// TwinCAT 3 PLC project SYC
// ProgramVersion: 3.1.4023.0
// libraries:
//   Tc2_Standard, * (Beckhoff Automation GmbH)
//   Tc2_System, * (Beckhoff Automation GmbH)
//   Tc2_Utilities, * (Beckhoff Automation GmbH)
//   Tc3_JsonXml, * (Beckhoff Automation GmbH)
//   Tc3_Module, * (Beckhoff Automation GmbH)
//   Base Interfaces,newest,System
// project tree:
//   / Class Diagram.TcCD (not stored), MAIN.TcPOU, PlcTask.TcTTO, Testing.TcPOU
//   Collection/ HashMap.TcPOU, Map.TcIO, MutableArray.TcPOU, List.TcIO, ListLength.TcDUT (not stored), ListType.TcDUT
//   Condition/ CResult.TcDUT, Is.TcPOU
//   Misc/ AddLeadingZeros.TcPOU, BaseConnector.TcPOU, CHAR.TcDUT, CONSTANTS.TcGVL, WCHAR.TcDUT, P2CHAR.TcPOU, P2WCHAR.TcPOU
//   Sequencer/ Condition.TcPOU, Sequencer.TcPOU, StepAction.TcDUT, StepCondition.TcDUT, StepTransition.TcDUT, Transition.TcPOU
//   Sequencer/WIP/ ConditionConfig.TcDUT (not stored), CurrentStep.TcDUT (not stored), E_Result.TcTLEO, StepConfig.TcDUT, StepLog.TcDUT, StepStatus.TcDUT
//   Signal/ Signal.TcPOU, SignalBundle.TcPOU, SignalMapping.TcDUT, SignalProvider.TcPOU, SignalTimer.TcDUT
//   SimpleStepLogger/ SimpleStepLog.TcDUT, SimpleStepLogger.TcPOU
//   SymbolProvider/ Symbol.TcDUT, SymbolProvider.TcPOU, SymbolProvider_1.TcPOU
//   Tools/ CallThisSingleTimeEachCycle.TcPOU, TaskHeartbeat.TcPOU, Regex.TcPOU, RegexMatch.TcDUT, System.TcPOU, SystemBundle.TcPOU, WRegex.TcPOU, TimeProvider.TcPOU
// real-time tasks:
//   TASK PlcTask: cycle T#10ms, priority 20, ADS port 350

CONFIGURATION SYC
    RESOURCE PLC ON TwinCAT3
        TASK PlcTask(INTERVAL := T#10ms, PRIORITY := 20);
        PROGRAM MAIN WITH PlcTask : MAIN;
        PROGRAM Testing WITH PlcTask : Testing;
    END_RESOURCE
END_CONFIGURATION

// ---- Condition/CResult.TcDUT
TYPE CResult :
STRUCT
	datatype	: INT;
	result		: BOOL;
END_STRUCT
END_TYPE

// ---- Collection/ListType.TcDUT

TYPE ListType :
STRUCT
	size			: UDINT;
	class			: __SYSTEM.TYPE_CLASS;
//	classPointer	: POINTER TO BYTE; // pointer to FB
	name			: T_MaxString;

	
	(*
	IDEA:
	if __SYSTEM.TYPE_CLASS <> USER_DEF then //int, bool, string
		classNumber := __SYSTEM.TYPE_CLASS
	else // function block
		classNumber := ADR(type)
		
	problems:
	 - how to achieve this in some user firendly way
	 - how to keep datatype pointer up to date after online change
	*)
//	classNumber		: UXINT; 

END_STRUCT
END_TYPE

// ---- Misc/CHAR.TcDUT
TYPE CHAR : STRING(1); END_TYPE

// ---- Misc/WCHAR.TcDUT
TYPE WCHAR : WSTRING(1); END_TYPE

// ---- Sequencer/StepAction.TcDUT
TYPE StepAction :
STRUCT
	name			: STRING;
	caseNumber		: INT;
//	timeout			: TIME;
//	timeoutAction	: STRING; these will go to binding
	description		: STRING;
END_STRUCT
END_TYPE

// ---- Sequencer/StepCondition.TcDUT
TYPE StepCondition :
STRUCT
	name			: STRING;
	condition		: Condition;
//	nextAction		: STRING;
//	timeout			: TIME;
//	timeoutAction	: STRING;
	/// these will go to binding
END_STRUCT
END_TYPE

// ---- Sequencer/StepTransition.TcDUT
TYPE StepTransition :
STRUCT
	actionName		: STRING;
	conditionName	: STRING;
	nextActionName	: STRING;
END_STRUCT
END_TYPE

// ---- Sequencer/WIP/E_Result.TcTLEO
{attribute 'qualified_only'}
{attribute 'strict'}
TYPE E_Result :
(
	done,
	timeout,
	error,
	interrupt,
	stop
);
END_TYPE

// ---- Sequencer/WIP/StepConfig.TcDUT
TYPE StepConfig :
STRUCT
	number		: INT;
	timeout		: TIME;
	
	description	: STRING;
END_STRUCT
END_TYPE

// ---- Sequencer/WIP/StepLog.TcDUT
TYPE StepLog :
STRUCT
	config 		: StepConfig;
	status		: StepStatus;
END_STRUCT
END_TYPE

// ---- Sequencer/WIP/StepStatus.TcDUT
TYPE StepStatus :
STRUCT
	status		: E_Result;
	elapsedTime : TIME;
END_STRUCT
END_TYPE

// ---- Signal/SignalMapping.TcDUT
TYPE SignalMapping :
STRUCT
	symbol	: POINTER TO BOOL;
	signal	: POINTER TO SignalBundle;
END_STRUCT
END_TYPE

// ---- Signal/SignalTimer.TcDUT

// Basically just timer IO with IN input excluded as it binded to the signal variable
TYPE SignalTimer :
STRUCT
	PT		: REFERENCE TO TIME;
	
	ET		: REFERENCE TO TIME;
	Q		: REFERENCE TO BOOL;
END_STRUCT
END_TYPE

// ---- SimpleStepLogger/SimpleStepLog.TcDUT
TYPE SimpleStepLog :
STRUCT
	number			: LINT;
	name			: STRING;
	description		: T_MaxString;
	duration		: TIME;
	mode			: STRING;
END_STRUCT
END_TYPE

// ---- SymbolProvider/Symbol.TcDUT
TYPE Symbol :
STRUCT
	info : __SYSTEM.AnyType; // varinfo?
	
	description : STRING;
END_STRUCT
END_TYPE

// ---- Tools/RegexMatch.TcDUT
TYPE RegexMatch :
STRUCT
	found : BOOL;
	start : INT;
	length : INT;
	text : STRING;
END_STRUCT
END_TYPE

// ---- Misc/CONSTANTS.TcGVL
VAR_GLOBAL CONSTANT
	MAX_DWORD	: DWORD := 4294967295;
	MAX_DWORD_2	: DWORD := -1;
	MAX_TIME	: TIME := TO_TIME(MAX_DWORD);
END_VAR

// ---- Collection/Map.TcIO

INTERFACE Map


METHOD Get : BOOL
VAR_INPUT
	
END_VAR
END_METHOD


METHOD Put : Map
VAR_INPUT
	key			: ANY;
	value		: ANY;
END_VAR
END_METHOD


METHOD Remove : Map
VAR_INPUT
END_VAR
END_METHOD


METHOD RemoveAll : Map
VAR_INPUT
END_VAR
END_METHOD

END_INTERFACE

// ---- Collection/List.TcIO

INTERFACE List


METHOD Append : List
VAR_INPUT
	data	: ANY;
END_VAR
END_METHOD


PROPERTY Datatype : ListType
GET
END_GET
END_PROPERTY

PROPERTY DatatypeDefined : BOOL
GET
END_GET
END_PROPERTY


// Delete pointers
METHOD FB_exit : BOOL
VAR_INPUT
	bInCopyCode : BOOL; // if TRUE, the exit method is called for exiting an instance that is copied afterwards (online change).
END_VAR
END_METHOD


METHOD Get : BOOL
VAR_INPUT
	index		: INT; // Allow for indexing from end
	destination	: ANY;
END_VAR
END_METHOD


METHOD Insert : List
VAR_INPUT
	index	: INT; // Allow for indexing from end
	data	: ANY;
END_VAR
END_METHOD


METHOD IsEmpty : BOOL
VAR_INPUT
END_VAR
END_METHOD


METHOD IsTypeCorrect : BOOL
VAR_INPUT
	checkedVariable		: ANY;
END_VAR
END_METHOD


PROPERTY LastIndex : ListLength
GET
END_GET
END_PROPERTY


PROPERTY Length : ListLength
GET
END_GET
END_PROPERTY


METHOD Prepend : List
VAR_INPUT
	data	: ANY;
END_VAR
END_METHOD


METHOD Remove : List
VAR_INPUT
	index	: INT; // Allow for indexing from end
END_VAR
END_METHOD


METHOD RemoveAll : List
VAR_INPUT
END_VAR
END_METHOD


METHOD Set : List
VAR_INPUT
	index	: INT; // Allow for indexing from end
	data	: ANY;
END_VAR
END_METHOD

END_INTERFACE

// ---- MAIN.TcPOU
PROGRAM MAIN
VAR
	sensor1 : BOOL;
	sensor2 : BOOL;
	sensor3 : BOOL;
	counter1 : INT;
	
	seq : Sequencer;
	firstCycle : BOOL := TRUE;
	test : BOOL;
	ceres : CResult;
	n1 : PVOID;
	n2 : PVOID;
	n3 : PVOID;
	
	re : Regex;
END_VAR

IF firstCycle THEN
	firstCycle := FALSE;
	
	RegisterActions();
	
END_IF

seq();

CASE seq.currentAction.caseNumber OF
	0 : // action code 1
	10 : // action code 2
	20 : // action code 3
	30 : // action code 4

END_CASE

Is(test);
Is(ceres);

n1 := SIZEOF(CResult);
n2 := SIZEOF(CResult.result);
n3 := SIZEOF(CResult.datatype);

re.match(pattern := 'he.*o', text := 'hellQQllo_HelloWorld').found;

ACTION RegisterActions:
//seq.ClearActions();

//seq.RegisterAction(
//	name := 'name 1',
//	number := 0
//);
//seq.RegisterAction(
//	name := 'name 2',
//	number := 10
//);
//seq.RegisterAction(
//	name := 'name 3',
//	number := 20
//);
//seq.RegisterAction(
//	name := 'name 4',
//	number := 30
//);
END_ACTION

ACTION RegisterAll:
// Register actions
seq.RegisterAction(
	name := 'name 1',
	caseNumber := 0,
	''
);
seq.RegisterAction(
	name := 'name 2',
	caseNumber := 10,
	''
);
seq.RegisterAction(
	name := 'name 3',
	caseNumber := 20,
	''
);
seq.RegisterAction(
	name := 'name 4',
	caseNumber := 30,
	''
);

// Register conditions
seq.RegisterCondition('cond 1').Is(sensor1);
seq.RegisterCondition('cond 2').Is(sensor2).AndIs(sensor3);
seq.RegisterCondition('cond 3').Is(sensor3);
seq.RegisterCondition('cond 4').Is(sensor3);

// Bind them together
seq.Bind('name 1')
	.WhenGoTo('cond 1', 'name 2');
seq.Bind('name 2')
	.WhenGoTo('cond 2', 'name 3')
	.WhenGoTo('cond 3', 'name 4');
seq.Bind('name 3')
	.WhenGoTo('cond 3', 'name 4');
seq.Bind('name 4')
	.WhenGoTo('cond 4', 'name 1');
END_ACTION

ACTION RegisterConditions:
//seq.ClearConditions();

//seq.RegisterCondition('cond 1').Is(sensor1);
//seq.RegisterCondition('cond 2').Is(sensor2).AndIs(sensor3);
//seq.RegisterCondition('cond 3').Is(sensor3);
//seq.RegisterCondition('cond 4').Is(sensor3);
END_ACTION

ACTION RegisterTransitions:
//seq.Bind('name 1')
//	.WhenGoTo('cond 1', 'name 2');
//seq.Bind('name 2')
//	.WhenGoTo('cond 2', 'name 3')
//	.WhenGoTo('cond 3', 'name 4');
//seq.Bind('name 3')
//	.WhenGoTo('cond 3', 'name 4');
//seq.Bind('name 4')
//	.WhenGoTo('cond 4', 'name 1');
END_ACTION

END_PROGRAM

// ---- Sequencer/Sequencer.TcPOU
FUNCTION_BLOCK Sequencer EXTENDS BaseConnector
VAR_INPUT
END_VAR
VAR_OUTPUT
END_VAR
VAR
	actions		: ARRAY[0..MAX_ACTION] OF StepAction;
	lastAction 	: INT := 0;
	currentAction : StepAction;
	startAction	: STRING;
	
	conditions	: ARRAY[0..MAX_CONDITION] OF StepCondition;
	lastCondition : INT := 0;
	currentCondition : StepCondition;
	
	timer		: TON := (PT := MAX_TIME);
	
END_VAR
VAR CONSTANT
	MAX_ACTION	: INT := 99;
	MAX_CONDITION : INT := 99;
END_VAR


timer(IN := TRUE);

//IF currentCondition.condition.satisfied THEN
	
//	ChangeStep(currentCondition.nextAction);
//ELSIF currentAction.timeout > T#0S AND_THEN timer.ET > currentAction.timeout THEN
	
//	ChangeStep(currentAction.timeoutAction);
//ELSIF currentCondition.timeout > T#0S AND_THEN timer.ET > currentCondition.timeout THEN

//	ChangeStep(currentCondition.timeoutAction);
//END_IF

METHOD Bind : REFERENCE TO Transition
VAR_INPUT
	actionName	: STRING;
END_VAR
END_METHOD

METHOD ChangeStep : BOOL
VAR_INPUT
	actionName		: STRING;
END_VAR
VAR
	i : INT;
END_VAR
//LogChange(currentAction.name, Condition, actionName);

FOR i := 0 TO MAX_ACTION DO
	IF (actions[i].name = actionName) THEN
		
		currentAction := actions[i];
	END_IF
END_FOR

timer(IN := FALSE);
timer(IN := TRUE);
END_METHOD

METHOD PRIVATE LogChange : BOOL
VAR_INPUT
	oldAction : STRING;
	satisfiedCondition : Condition;
	nextAction : STRING;
END_VAR
// TODO
END_METHOD

METHOD RegisterAction : BOOL
VAR_INPUT
	name			: STRING;
	caseNumber		: INT;
	description		: STRING;
END_VAR
VAR
	a : REFERENCE TO StepAction REF= actions[lastAction];
END_VAR
a.name := name;
a.caseNumber := caseNumber;
//a.timeout := timeout;
//a.timeoutAction := timeoutAction;
a.description := description;

lastAction := lastAction + 1;
END_METHOD

METHOD RegisterCondition : REFERENCE TO Condition
VAR_INPUT
	name			: STRING;
END_VAR
VAR
	c : REFERENCE TO StepCondition REF= conditions[lastAction];
END_VAR
c.name := name;
//c.condition := condition;
//c.nextAction := nextAction;
//c.timeout := timeout;
//c.timeoutAction := timeoutAction;

lastCondition := lastCondition + 1;

RegisterCondition REF= c.condition;
END_METHOD

METHOD Start : BOOL
VAR_INPUT
	startAction		: STRING;
END_VAR
THIS^.startAction := startAction; 

ChangeStep(startAction);
END_METHOD

END_FUNCTION_BLOCK

// ---- Misc/BaseConnector.TcPOU
FUNCTION_BLOCK BaseConnector
VAR_INPUT
END_VAR
VAR_OUTPUT
END_VAR
VAR
END_VAR
VAR_STAT
	sp	: SymbolProvider;
END_VAR

END_FUNCTION_BLOCK

// ---- SymbolProvider/SymbolProvider.TcPOU
FUNCTION_BLOCK SymbolProvider
VAR_INPUT
END_VAR
VAR_OUTPUT
END_VAR
VAR
	list : ARRAY[0..99] OF Symbol;
	lastIndex : UINT := 0;
END_VAR

METHOD Get : STRING
VAR_INPUT
	symbol : ANY;
END_VAR
VAR
	i : UINT;
END_VAR
FOR i := 0 TO lastIndex DO
	IF symbol.pValue = list[i].info.pValue THEN
		Get := list[i].description;
		RETURN;
	END_IF
END_FOR
END_METHOD

METHOD Register : BOOL
VAR_INPUT
	symbol				: ANY;
	descriptionName		: STRING;
END_VAR
list[lastIndex].info := symbol;
list[lastIndex].description := descriptionName;
END_METHOD

END_FUNCTION_BLOCK

// ---- Sequencer/Transition.TcPOU
FUNCTION_BLOCK Transition
VAR_INPUT
END_VAR
VAR_OUTPUT
END_VAR
VAR
END_VAR

METHOD WhenGoTo : reference TO Transition
VAR_INPUT
	conditionName	: STRING;
	nextActionName	: STRING;
END_VAR
END_METHOD

END_FUNCTION_BLOCK

// ---- Sequencer/Condition.TcPOU
FUNCTION_BLOCK Condition EXTENDS BaseConnector
VAR_INPUT
END_VAR
VAR_OUTPUT
END_VAR
VAR
	config		: ARRAY[0..99] OF ConditionConfig;
	result		: BOOL;
END_VAR

METHOD AndIs : REFERENCE TO Condition
VAR_INPUT
	symbol	: ANY;
END_VAR
END_METHOD

METHOD AndIsNot : Condition
VAR_INPUT
END_VAR
END_METHOD

METHOD Is : REFERENCE TO Condition
VAR_INPUT
	symbol	: ANY;
END_VAR
END_METHOD

METHOD IsNot : Condition
VAR_INPUT
END_VAR
END_METHOD

METHOD OrIs : Condition
VAR_INPUT
END_VAR
END_METHOD

METHOD OrIsNot : Condition
VAR_INPUT
END_VAR
END_METHOD

PROPERTY satisfied : BOOL
GET
END_GET
END_PROPERTY

END_FUNCTION_BLOCK

// ---- Condition/Is.TcPOU
FUNCTION Is : CResult
VAR_INPUT
	symbol		: ANY;
END_VAR
VAR
	typeReader	: FB_JsonReadWriteDatatype;
	t : STRING;
END_VAR

CASE symbol.TypeClass OF
	
	IBaseLibrary.TypeClass.TYPE_BOOL:

		Is.result := PBOOL_TO_BOOL(symbol.pValue);
		Is.datatype := TO_INT(symbol.TypeClass);
		
	IBaseLibrary.TypeClass.TYPE_USERDEF:
		IF typeReader.GetDatatypeNameByAddress(pData := symbol.pValue, nData := symbol.diSize) = 'CResult' THEN

			Is.result := PBOOL_TO_BOOL(symbol.pValue + ADR(Is.result) - ADR(Is));
			Is.datatype := 420;
		END_IF

END_CASE

END_FUNCTION

// ---- Tools/Regex.TcPOU
FUNCTION_BLOCK Regex
VAR_INPUT
END_VAR
VAR_OUTPUT
END_VAR
VAR
	result : RegexMatch;
END_VAR

//https://stackoverflow.com/questions/4040835/how-do-i-write-a-simple-regular-expression-pattern-matching-function-in-c-or-c

METHOD incMatchPos : BOOL
VAR_INPUT
	isMatch : BOOL;
END_VAR
IF isMatch THEN
	result.length := result.length + 1;
ELSE
	result.start := result.start + 1;
	result.length := 0;
END_IF
incMatchPos := isMatch;
END_METHOD

METHOD match : REFERENCE TO RegexMatch
VAR_INPUT
	pattern : STRING;
	text	: STRING;
END_VAR
result.start := 1;
result.length := 0;
result.found := matchP(ADR(pattern), ADR(text));
result.text := MID(STR := text, POS := result.start, LEN := result.length);

match REF= result;
END_METHOD

METHOD PRIVATE matchHere : BOOL
VAR_INPUT
	pattern : POINTER TO STRING;
	text	: POINTER TO STRING;
END_VAR
IF P2CHAR(pattern) = '$00' THEN
	matchHere := TRUE;
	RETURN;
ELSIF P2CHAR(pattern + 1) = '*' THEN
	matchHere := matchStar(P2CHAR(pattern), pattern + 2, text);
	RETURN;
ELSIF P2CHAR(pattern) = '$$' AND P2CHAR(pattern + 1) = '$00' THEN
	matchHere := P2CHAR(text) = '$00';
	RETURN;
ELSIF text^ <> '$00' AND (P2CHAR(pattern) = '.' OR P2CHAR(pattern) = P2CHAR(text)) THEN
	matchHere := THIS^.matchHere(pattern + 1, text + 1);
	incMatchPos(matchHere);
	RETURN;
END_IF



///* matchhere: search FOR regexp AT beginning OF text */
//int matchhere(char *regexp, char *text)
//{
//    if (regexp[0] == '\0')
//        return 1;
//    if (regexp[1] == '*')
//        return matchstar(regexp[0], regexp+2, text);
//    if (regexp[0] == '$' && regexp[1] == '\0')
//        return *text == '\0';
//    if (*text!='\0' && (regexp[0]=='.' || regexp[0]==*text))
//        return matchhere(regexp+1, text+1);
//    return 0;
//}
END_METHOD

METHOD matchP : BOOL
VAR_INPUT
	pattern : POINTER TO STRING;
	text	: POINTER TO STRING;
END_VAR
IF P2CHAR(pattern) = '^' THEN
	matchP := matchHere(pattern + 1, text);
	RETURN;
END_IF
REPEAT
	IF matchHere(pattern, text) THEN
		matchP := TRUE;
		RETURN;
	END_IF
UNTIL
	NOT(P2CHAR(text) <> '$00') AND (text := text + 1) <> NULL AND (incMatchPos(matchP) OR TRUE) //pointer dereference and increment oneliner
END_REPEAT



///* match: search FOR regexp anywhere in text */
//int match(char *regexp, char *text)
//{
//    if (regexp[0] == '^')
//        return matchhere(regexp+1, text);
//    do {    /* must look even if string is empty */
//        if (matchhere(regexp, text))
//            return 1;
//    } while (*text++ != '\0');
//    return 0;
//}
END_METHOD

METHOD PRIVATE matchStar : BOOL
VAR_INPUT
	c		: CHAR;
	pattern : POINTER TO STRING;
	text	: POINTER TO STRING;
END_VAR
REPEAT
	IF matchHere(pattern, text) THEN
		matchStar := TRUE;
		RETURN;
	END_IF
UNTIL
	NOT(P2CHAR(text) <> '$00' AND (P2CHAR(text) = c OR c = '.')) AND (text := text + 1) > null AND (incMatchPos(NOT matchStar) OR TRUE)
END_REPEAT


///* matchstar: search FOR c*regexp AT beginning OF text */
//int matchstar(int c, char *regexp, char *text)
//{
//    do {    /* a * matches zero or more instances */
//        if (matchhere(regexp, text))
//            return 1;
//    } while (*text != '\0' && (*text++ == c || c == '.'));
//    return 0;
//}
END_METHOD

END_FUNCTION_BLOCK

// ---- Misc/P2CHAR.TcPOU
FUNCTION P2CHAR : CHAR
VAR_INPUT
	p : POINTER TO STRING;
END_VAR
VAR
END_VAR

P2CHAR := p^;

END_FUNCTION

// ---- Testing.TcPOU
PROGRAM Testing
VAR
	test		: STRING := 'ahoj';
	byteContent	: ARRAY[1..SIZEOF(test)] OF BYTE;
	
	beat : BOOL;
	t : STRING;
END_VAR

test := TO_STRING(ADR(byteContent));

CallThisSingleTimeEachCycle();


beat := System().GetTaskHeartbeat();
t := System().TimeProvider.GetTimeString('{h}:{m}:{s},{S}');

END_PROGRAM

// ---- Tools/CallThisSingleTimeEachCycle.TcPOU

FUNCTION CallThisSingleTimeEachCycle : BOOL


TaskHeartbeat(update := TRUE);

END_FUNCTION

// ---- Tools/TaskHeartbeat.TcPOU

FUNCTION TaskHeartbeat : BOOL;
VAR_INPUT
	update		: BOOL;
END_VAR
VAR_STAT
	_beat		: BOOL;
END_VAR


IF (update) THEN
	_beat := NOT _beat;
END_IF

TaskHeartbeat := _beat;

END_FUNCTION

// ---- Tools/System.TcPOU

FUNCTION System : REFERENCE TO SystemBundle
VAR_INPUT
END_VAR
VAR
	bundle		: SystemBundle;
END_VAR


bundle.Call();

System REF= bundle;

END_FUNCTION

// ---- Tools/SystemBundle.TcPOU

FUNCTION_BLOCK SystemBundle
VAR_INPUT
END_VAR
VAR_OUTPUT
END_VAR
VAR
	_timeProvider		: TimeProvider;
END_VAR

METHOD Call : BOOL
VAR_INPUT
END_VAR

_timeProvider();
END_METHOD


METHOD GetTaskHeartbeat : BOOL
VAR_INPUT
END_VAR

GetTaskHeartbeat := TaskHeartbeat(update := FALSE);
END_METHOD

PROPERTY TimeProvider : REFERENCE TO TimeProvider
GET

TimeProvider REF= _timeProvider;
END_GET
END_PROPERTY

END_FUNCTION_BLOCK

// ---- Tools/TimeProvider.TcPOU
FUNCTION_BLOCK TimeProvider
VAR_INPUT
END_VAR
VAR_OUTPUT
END_VAR
VAR
	localSystemTime						: FB_LocalSystemTime;
	
	// timestamp
	getTimeZoneInformation 			: FB_GetTimeZoneInformation;
    timeZoneInformation 			: ST_TimeZoneInformation;
    specificLocalTimeToFileTime 	: FB_TzSpecificLocalTimeToFileTime;
    fileTime						: T_FILETIME;
    onZerothSecondLastCycle 		: BOOL;
END_VAR

localSystemTime(bEnable := FALSE);


//https://stackoverflow.com/questions/41773732/how-do-i-get-the-unix-timestamp-in-twincat3

// On the zeroth second of each minutesync timezone information
IF (timeZoneInformation.standardName = '' OR (localSystemTime.systemTime.wSecond = 0 AND NOT onZerothSecondLastCycle)) THEN
    getTimeZoneInformation(sNetID := '', bExecute := TRUE, tzInfo => timeZoneInformation);
END_IF;

// Convert local system time to unix timestamps
specificLocalTimeToFileTime(in := Tc2_Utilities.SYSTEMTIME_TO_FILETIME(localSystemTime.systemTime), tzInfo := timeZoneInformation, out => fileTime);
//seconds := (SHL(DWORD_TO_ULINT(fileTime.dwHighDateTime), 32) + DWORD_TO_ULINT(fileTime.dwLowDateTime)) / 10000000 - 11644473600;
//milliseconds := (SHL(DWORD_TO_ULINT(fileTime.dwHighDateTime), 32) + DWORD_TO_ULINT(fileTime.dwLowDateTime)) / 10000 - 11644473600000;

onZerothSecondLastCycle := localSystemTime.systemTime.wSecond = 0;

METHOD FB_init : BOOL
VAR_INPUT
	bInitRetains : BOOL; // if TRUE, the retain variables are initialized (warm start / cold start)
	bInCopyCode : BOOL;  // if TRUE, the instance afterwards gets moved into the copy code (online change)
END_VAR
localSystemTime(bEnable := TRUE);
END_METHOD

METHOD GetMonthName : STRING
VAR_INPUT
	monthNumber			: UINT;
	shortName			: BOOL;
END_VAR
IF shortName THEN
	CASE monthNumber OF
		1	: GetMonthName := 'Jan';
		2	: GetMonthName := 'Feb';
		3	: GetMonthName := 'Mar';
		4	: GetMonthName := 'Apr';
		5	: GetMonthName := 'May';
		6	: GetMonthName := 'Jun';
		7	: GetMonthName := 'Jul';
		8	: GetMonthName := 'Aug';
		9	: GetMonthName := 'Sep';
		10	: GetMonthName := 'Oct';
		11	: GetMonthName := 'Nov';
		12	: GetMonthName := 'Dec';
	END_CASE
ELSE
	CASE monthNumber OF
		1	: GetMonthName := 'January';
		2	: GetMonthName := 'February';
		3	: GetMonthName := 'March';
		4	: GetMonthName := 'April';
		5	: GetMonthName := 'May';
		6	: GetMonthName := 'June';
		7	: GetMonthName := 'July';
		8	: GetMonthName := 'August';
		9	: GetMonthName := 'September';
		10	: GetMonthName := 'October';
		11	: GetMonthName := 'November';
		12	: GetMonthName := 'December';
	END_CASE
END_IF
END_METHOD

METHOD GetTimeString : STRING
VAR_INPUT
	format : STRING; //hh:mm:ss:SSS dd:MM:yyyy https://www.ibm.com/docs/en/rtw/9.0.1?topic=reference-formatting-parsing-date-time-patterns
END_VAR
VAR
	placeholder : STRING(4);
	
	beginIndex	: INT;
	endIndex	: INT;
	length		: INT;
		
END_VAR
GetTimeString := format;

WHILE (beginIndex := FIND(GetTimeString, '{')) > 0 AND (endIndex := FIND(GetTimeString, '}')) > (beginIndex + 1) AND  (length := endIndex - beginIndex - 1) > 0 DO
	
	placeholder := MID(STR := GetTimeString, POS := beginIndex + 1, LEN := length);
		
	IF 		placeholder = 'h' 		THEN GetTimeString := REPLACE( STR1 := GetTimeString, STR2 := TO_STRING(localSystemTime.systemTime.wHour), L := length + 2, P := beginIndex);
	ELSIF 	placeholder = 'hh' 		THEN GetTimeString := REPLACE( STR1 := GetTimeString, STR2 := AddLeadingZeros(TO_STRING(localSystemTime.systemTime.wHour), 2), L := length + 2, P := beginIndex);
	ELSIF 	placeholder = 'm' 		THEN GetTimeString := REPLACE( STR1 := GetTimeString, STR2 := TO_STRING(localSystemTime.systemTime.wMinute), L := length + 2, P := beginIndex);
	ELSIF 	placeholder = 'mm' 		THEN GetTimeString := REPLACE( STR1 := GetTimeString, STR2 := AddLeadingZeros(TO_STRING(localSystemTime.systemTime.wMinute), 2), L := length + 2, P := beginIndex);
	ELSIF 	placeholder = 's' 		THEN GetTimeString := REPLACE( STR1 := GetTimeString, STR2 := TO_STRING(localSystemTime.systemTime.wSecond), L := length + 2, P := beginIndex);
	ELSIF 	placeholder = 'ss' 		THEN GetTimeString := REPLACE( STR1 := GetTimeString, STR2 := AddLeadingZeros(TO_STRING(localSystemTime.systemTime.wSecond), 2), L := length + 2, P := beginIndex);
	ELSIF 	placeholder = 'S' 		THEN GetTimeString := REPLACE( STR1 := GetTimeString, STR2 := TO_STRING(localSystemTime.systemTime.wMilliseconds/100), L := length + 2, P := beginIndex);
	ELSIF 	placeholder = 'SS' 		THEN GetTimeString := REPLACE( STR1 := GetTimeString, STR2 := AddLeadingZeros(TO_STRING(localSystemTime.systemTime.wMilliseconds/10), 2), L := length + 2, P := beginIndex);
	ELSIF 	placeholder = 'SSS' 	THEN GetTimeString := REPLACE( STR1 := GetTimeString, STR2 := AddLeadingZeros(TO_STRING(localSystemTime.systemTime.wMilliseconds), 3), L := length + 2, P := beginIndex);
	ELSIF 	placeholder = 'd' 		THEN GetTimeString := REPLACE( STR1 := GetTimeString, STR2 := TO_STRING(localSystemTime.systemTime.wDay), L := length + 2, P := beginIndex);
	ELSIF 	placeholder = 'dd' 		THEN GetTimeString := REPLACE( STR1 := GetTimeString, STR2 := AddLeadingZeros(TO_STRING(localSystemTime.systemTime.wDay), 2), L := length + 2, P := beginIndex);
	ELSIF 	placeholder = 'ddd' 	THEN GetTimeString := REPLACE( STR1 := GetTimeString, STR2 := GetWeekdayName(localSystemTime.systemTime.wDayOfWeek, TRUE), L := length + 2, P := beginIndex);
	ELSIF 	placeholder = 'dddd'	THEN GetTimeString := REPLACE( STR1 := GetTimeString, STR2 := GetWeekdayName(localSystemTime.systemTime.wDayOfWeek, FALSE), L := length + 2, P := beginIndex);
	ELSIF 	placeholder = 'M' 		THEN GetTimeString := REPLACE( STR1 := GetTimeString, STR2 := TO_STRING(localSystemTime.systemTime.wMonth), L := length + 2, P := beginIndex);
	ELSIF 	placeholder = 'MM' 		THEN GetTimeString := REPLACE( STR1 := GetTimeString, STR2 := AddLeadingZeros(TO_STRING(localSystemTime.systemTime.wMonth), 2), L := length + 2, P := beginIndex);
	ELSIF 	placeholder = 'MMM' 	THEN GetTimeString := REPLACE( STR1 := GetTimeString, STR2 := GetMonthName(localSystemTime.systemTime.wMonth, TRUE), L := length + 2, P := beginIndex);
	ELSIF 	placeholder = 'MMMM'	THEN GetTimeString := REPLACE( STR1 := GetTimeString, STR2 := GetMonthName(localSystemTime.systemTime.wMonth, FALSE), L := length + 2, P := beginIndex);
	ELSIF 	placeholder = 'y' OR placeholder = 'yy' OR placeholder = 'yyy' OR placeholder = 'yyyy'
									THEN GetTimeString := REPLACE( STR1 := GetTimeString, STR2 := RIGHT(TO_STRING(localSystemTime.systemTime.wYear), length), L := length + 2, P := beginIndex);
	ELSE 
			GetTimeString := REPLACE( STR1 := GetTimeString, STR2 := 'ERR', L := length + 2, P := beginIndex);
	END_IF
END_WHILE
END_METHOD

// deprecated. Use optimized GetTimeString() instead
METHOD GetTimeStringRe : STRING
VAR_INPUT
	format : STRING; //hh:mm:ss:SSS dd:MM:yyyy https://www.ibm.com/docs/en/rtw/9.0.1?topic=reference-formatting-parsing-date-time-patterns
END_VAR
VAR
	re : Regex;
	placeholder : STRING(4);
END_VAR
GetTimeStringRe := format;

WHILE re.match('{.*}', GetTimeStringRe).found DO
	placeholder := MID(STR := re.result.text, POS := 2, LEN := re.result.length - 2);
	
	IF 		placeholder = 'h' 		THEN GetTimeStringRe := REPLACE( STR1 := GetTimeStringRe, STR2 := TO_STRING(localSystemTime.systemTime.wHour), L := re.result.length, P := re.result.start);
	ELSIF 	placeholder = 'hh' 		THEN GetTimeStringRe := REPLACE( STR1 := GetTimeStringRe, STR2 := AddLeadingZeros(TO_STRING(localSystemTime.systemTime.wHour), 2), L := re.result.length, P := re.result.start);
	ELSIF 	placeholder = 'm' 		THEN GetTimeStringRe := REPLACE( STR1 := GetTimeStringRe, STR2 := TO_STRING(localSystemTime.systemTime.wMinute), L := re.result.length, P := re.result.start);
	ELSIF 	placeholder = 'mm' 		THEN GetTimeStringRe := REPLACE( STR1 := GetTimeStringRe, STR2 := AddLeadingZeros(TO_STRING(localSystemTime.systemTime.wMinute), 2), L := re.result.length, P := re.result.start);
	ELSIF 	placeholder = 's' 		THEN GetTimeStringRe := REPLACE( STR1 := GetTimeStringRe, STR2 := TO_STRING(localSystemTime.systemTime.wSecond), L := re.result.length, P := re.result.start);
	ELSIF 	placeholder = 'ss' 		THEN GetTimeStringRe := REPLACE( STR1 := GetTimeStringRe, STR2 := AddLeadingZeros(TO_STRING(localSystemTime.systemTime.wSecond), 2), L := re.result.length, P := re.result.start);
	ELSIF 	placeholder = 'S' 		THEN GetTimeStringRe := REPLACE( STR1 := GetTimeStringRe, STR2 := TO_STRING(localSystemTime.systemTime.wMilliseconds/100), L := re.result.length, P := re.result.start);
	ELSIF 	placeholder = 'SS' 		THEN GetTimeStringRe := REPLACE( STR1 := GetTimeStringRe, STR2 := AddLeadingZeros(TO_STRING(localSystemTime.systemTime.wMilliseconds/10), 2), L := re.result.length, P := re.result.start);
	ELSIF 	placeholder = 'SSS' 	THEN GetTimeStringRe := REPLACE( STR1 := GetTimeStringRe, STR2 := AddLeadingZeros(TO_STRING(localSystemTime.systemTime.wMilliseconds), 3), L := re.result.length, P := re.result.start);
	ELSIF 	placeholder = 'd' 		THEN GetTimeStringRe := REPLACE( STR1 := GetTimeStringRe, STR2 := TO_STRING(localSystemTime.systemTime.wDay), L := re.result.length, P := re.result.start);
	ELSIF 	placeholder = 'dd' 		THEN GetTimeStringRe := REPLACE( STR1 := GetTimeStringRe, STR2 := AddLeadingZeros(TO_STRING(localSystemTime.systemTime.wDay), 2), L := re.result.length, P := re.result.start);
	ELSIF 	placeholder = 'ddd' 	THEN GetTimeStringRe := REPLACE( STR1 := GetTimeStringRe, STR2 := GetWeekdayName(localSystemTime.systemTime.wDayOfWeek, TRUE), L := re.result.length, P := re.result.start);
	ELSIF 	placeholder = 'dddd'	THEN GetTimeStringRe := REPLACE( STR1 := GetTimeStringRe, STR2 := GetWeekdayName(localSystemTime.systemTime.wDayOfWeek, FALSE), L := re.result.length, P := re.result.start);
	ELSIF 	placeholder = 'M' 		THEN GetTimeStringRe := REPLACE( STR1 := GetTimeStringRe, STR2 := TO_STRING(localSystemTime.systemTime.wMonth), L := re.result.length, P := re.result.start);
	ELSIF 	placeholder = 'MM' 		THEN GetTimeStringRe := REPLACE( STR1 := GetTimeStringRe, STR2 := AddLeadingZeros(TO_STRING(localSystemTime.systemTime.wMonth), 2), L := re.result.length, P := re.result.start);
	ELSIF 	placeholder = 'MMM' 	THEN GetTimeStringRe := REPLACE( STR1 := GetTimeStringRe, STR2 := GetMonthName(localSystemTime.systemTime.wMonth, TRUE), L := re.result.length, P := re.result.start);
	ELSIF 	placeholder = 'MMMM'	THEN GetTimeStringRe := REPLACE( STR1 := GetTimeStringRe, STR2 := GetMonthName(localSystemTime.systemTime.wMonth, FALSE), L := re.result.length, P := re.result.start);
	ELSIF 	placeholder = 'y' OR placeholder = 'yy' OR placeholder = 'yyy' OR placeholder = 'yyyy'
									THEN GetTimeStringRe := REPLACE( STR1 := GetTimeStringRe, STR2 := RIGHT(TO_STRING(localSystemTime.systemTime.wYear), re.result.length - 2), L := re.result.length, P := re.result.start);
	ELSE 
			GetTimeStringRe := REPLACE( STR1 := GetTimeStringRe, STR2 := 'ERR', L := re.result.length, P := re.result.start);
	END_IF
END_WHILE
END_METHOD

METHOD GetWeekdayName : STRING
VAR_INPUT
	weekDayNumber		: UINT;
	shortName			: BOOL;
END_VAR
IF shortName THEN
	CASE weekDayNumber OF
		0	: GetWeekdayName := 'Sun';
		1	: GetWeekdayName := 'Mon';
		2	: GetWeekdayName := 'Tue';
		3	: GetWeekdayName := 'Wed';
		4	: GetWeekdayName := 'Thu';
		5	: GetWeekdayName := 'Fri';
		6	: GetWeekdayName := 'Sat';
	END_CASE
ELSE
	CASE weekDayNumber OF
		0	: GetWeekdayName := 'Sunday';
		1	: GetWeekdayName := 'Monday';
		2	: GetWeekdayName := 'Tuesday';
		3	: GetWeekdayName := 'Wednesday';
		4	: GetWeekdayName := 'Thursday';
		5	: GetWeekdayName := 'Friday';
		6	: GetWeekdayName := 'Saturday';
	END_CASE
END_IF
END_METHOD

PROPERTY Timestamp : ULINT // Unix timestamp in milliseconds
GET
// TODO is this even right?
Timestamp := (SHL(DWORD_TO_ULINT(fileTime.dwHighDateTime), 32) + DWORD_TO_ULINT(fileTime.dwLowDateTime)) / 10000 - 11644473600000;
END_GET
END_PROPERTY

PROPERTY TimeStruct : TIMESTRUCT // Week starts with Sunday
GET
TimeStruct := localSystemTime.systemTime;
END_GET
END_PROPERTY

PROPERTY TimeStructISO8601 : TIMESTRUCT // Week starts with Monday
GET
TimeStructISO8601 := localSystemTime.systemTime;
IF TimeStructISO8601.wDayOfWeek = 0 THEN
	TimeStructISO8601.wDayOfWeek := 6; // Move Sunday to the end of the week
ELSE
	TimeStructISO8601.wDayOfWeek := TimeStructISO8601.wDayOfWeek - 1;
END_IF
END_GET
END_PROPERTY

END_FUNCTION_BLOCK

// ---- Misc/AddLeadingZeros.TcPOU
FUNCTION AddLeadingZeros : STRING
VAR_INPUT
	str : STRING;
	charNumber : USINT;
END_VAR
VAR
END_VAR

AddLeadingZeros := str;
IF charNumber > LEN(str) THEN
	AddLeadingZeros := CONCAT('0', AddLeadingZeros);
	AddLeadingZeros := .AddLeadingZeros(AddLeadingZeros, charNumber);
END_IF

END_FUNCTION

// ---- Collection/HashMap.TcPOU

FUNCTION_BLOCK HashMap IMPLEMENTS Map
VAR_INPUT
END_VAR
VAR_OUTPUT
END_VAR
VAR
	//needs custom array handling instead of mutable array
	keys		:	MutableArray;
	values		: 	MutableArray;
END_VAR


METHOD Get : BOOL
VAR_INPUT
END_VAR
END_METHOD


METHOD Put : Map
VAR_INPUT
	key			: ANY;
	value		: ANY;
END_VAR

IF (((keys.DatatypeDefined AND values.DatatypeDefined) AND_THEN
	 (keys.IsTypeCorrect(key) AND values.IsTypeCorrect(value))) OR_ELSE
	(NOT keys.DatatypeDefined AND NOT values.DatatypeDefined)) THEN
	
	// needs hash function and custom array handling instead of mutable array
	keys.Append(key);
	values.Append(value);
END_IF
END_METHOD


METHOD Remove : Map
VAR_INPUT
END_VAR
END_METHOD


METHOD RemoveAll : Map
VAR_INPUT
END_VAR
END_METHOD

END_FUNCTION_BLOCK

// ---- Collection/MutableArray.TcPOU

{attribute 'hide_all_locals'}
FUNCTION_BLOCK MutableArray IMPLEMENTS List
VAR_INPUT
END_VAR
VAR_OUTPUT
END_VAR
VAR
	arr					: POINTER TO BYTE;
	_length				: ListLength;
	_datatype			: ListType;
	capacity			: ListLength;
	_datatypeDefined	: BOOL;
END_VAR
VAR CONSTANT
	GROWTH_FACTOR		: UDINT := 2;
	INITIAL_CAPACITY	: UDINT := 2;
END_VAR


METHOD PRIVATE Alloc : BOOL
VAR_INPUT
END_VAR
VAR
	allocSize	: UDINT;
END_VAR

capacity := INITIAL_CAPACITY;
allocSize := _datatype.size * capacity;
arr := __NEW(BYTE, allocSize);
END_METHOD


METHOD Append : List
VAR_INPUT
	data	: ANY;
END_VAR

Append := THIS^;

IF (NOT _datatypeDefined) THEN
	
	_datatype.size := TO_UDINT(data.diSize);
	_datatype.class := data.TypeClass;
	
	_datatypeDefined := TRUE;
	
	Alloc();
	
	MEMCPY(destAddr := arr + _length * _datatype.size, srcAddr := data.pValue, n := _datatype.size);

	_length := _length + 1;
ELSIF (IsTypeCorrect(data)) THEN
	
	IF (_length = capacity) THEN
		Grow();
	END_IF
	
	MEMCPY(destAddr := arr + _length * _datatype.size, srcAddr := data.pValue, n := _datatype.size);
	
	_length := _length + 1;
END_IF
END_METHOD


PROPERTY Datatype : ListType
GET

Datatype := _datatype;
END_GET
END_PROPERTY


PROPERTY DatatypeDefined : BOOL
GET

DatatypeDefined := _datatypeDefined;
END_GET
END_PROPERTY


// Delete pointers
METHOD FB_exit : BOOL
VAR_INPUT
	bInCopyCode : BOOL; // if TRUE, the exit method is called for exiting an instance that is copied afterwards (online change).
END_VAR

__DELETE(arr);
END_METHOD


METHOD Get : BOOL
VAR_INPUT
	index		: INT; // Allow for indexing from end
	destination	: ANY;
END_VAR
VAR
	arrIndex	: UDINT;
END_VAR

IF (_length = 0 OR NOT IsTypeCorrect(destination)) THEN
	RETURN;
END_IF

arrIndex := GetArrayIndex(index);

IF (IsArrayIndexValid(arrIndex)) THEN

	MEMCPY(destAddr := destination.pValue, srcAddr := arr + arrIndex * _datatype.size, n := _datatype.size);
END_IF
END_METHOD


METHOD PRIVATE GetArrayIndex : UDINT
VAR_INPUT
	index		: INT;
END_VAR

IF (index >= 0) THEN
	GetArrayIndex := TO_UDINT(index);
ELSE
	GetArrayIndex := _length + TO_UDINT(index);
END_IF
END_METHOD


METHOD PRIVATE Grow : BOOL
VAR_INPUT
END_VAR
VAR
	sizeToCopy		: UDINT;
	allocSize		: UDINT;
	newArr			: PVOID;
END_VAR

capacity := capacity * GROWTH_FACTOR;
allocSize := _datatype.size * capacity;
newArr := __NEW(BYTE, allocSize);

sizeToCopy := _datatype.size * _length; 
MEMCPY(destAddr := newArr, srcAddr := arr, n := sizeToCopy);

__DELETE(arr);
arr := newArr;
END_METHOD


METHOD Insert : List
VAR_INPUT
	index	: INT; // Allow for indexing from end
	data	: ANY;
END_VAR
VAR
	arrIndex	: UDINT;
	moveLength	: UDINT;
	indexAdr	: PVOID;
END_VAR

Insert := THIS^;

arrIndex := GetArrayIndex(index);

IF (NOT _datatypeDefined AND arrIndex = 0) THEN
	
	_datatype.size := TO_UDINT(data.diSize);
	_datatype.class := data.TypeClass;
	
	_datatypeDefined := TRUE;
	
	Alloc();
	
	MEMCPY(destAddr := arr + _length * _datatype.size, srcAddr := data.pValue, n := _datatype.size);

	_length := _length + 1;
ELSIF (IsTypeCorrect(data)) THEN
	IF (IsArrayIndexValid(arrIndex) OR _length = 0 OR arrIndex = _length) THEN

		IF (_length = capacity) THEN
			Grow();
		END_IF
		
		moveLength := _length - arrIndex;
		indexAdr := arr + arrIndex * _datatype.size;
		IF (moveLength > 0) THEN
			MEMMOVE(destAddr := indexAdr + _datatype.size, srcAddr := indexAdr, n := moveLength * _datatype.size);
		END_IF
		
		MEMCPY(destAddr := indexAdr, srcAddr := data.pValue, n := _datatype.size);
		
		_length := _length + 1;
	END_IF
END_IF
END_METHOD


METHOD PRIVATE IsArrayIndexValid : BOOL
VAR_INPUT
	arrIndex	: UDINT;
END_VAR

IsArrayIndexValid := arrIndex >= 0 AND arrIndex < _length;
END_METHOD


METHOD IsEmpty : BOOL
VAR_INPUT
END_VAR

IsEmpty := _length = 0;
END_METHOD


METHOD IsTypeCorrect : BOOL
VAR_INPUT
	checkedVariable		: ANY;
END_VAR

IsTypeCorrect :=
	checkedVariable.diSize = _datatype.size AND
	checkedVariable.TypeClass = _datatype.class;
END_METHOD


PROPERTY LastIndex : ListLength
GET

IF (_length = 0) THEN
	LastIndex := 0;
ELSE
	LastIndex := _length - 1;
END_IF
END_GET
END_PROPERTY


PROPERTY Length : ListLength
GET

Length := _length;
END_GET
END_PROPERTY


METHOD Prepend : List
VAR_INPUT
	data	: ANY;
END_VAR

Prepend := THIS^;

IF (NOT _datatypeDefined) THEN
	
	_datatype.size := TO_UDINT(data.diSize);
	_datatype.class := data.TypeClass;
	
	_datatypeDefined := TRUE;
	
	Alloc();
	
	MEMCPY(destAddr := arr + _length * _datatype.size, srcAddr := data.pValue, n := _datatype.size);

	_length := _length + 1;
ELSIF (IsTypeCorrect(data)) THEN
	
	IF (_length = capacity) THEN
		Grow();
	END_IF
	
	MEMMOVE(destAddr := arr + _datatype.size, srcAddr := arr, n := _length * _datatype.size);
	MEMCPY(destAddr := arr, srcAddr := data.pValue, n := _datatype.size);
	
	_length := _length + 1;
END_IF
END_METHOD


METHOD Remove : List
VAR_INPUT
	index		: INT; // Allow for indexing from end
END_VAR
VAR
	arrIndex	: UDINT;
	moveLength	: UDINT;
	indexAdr	: PVOID;
END_VAR

Remove := THIS^;

IF (_length = 0) THEN
	RETURN;
END_IF

arrIndex := GetArrayIndex(index);

IF (IsArrayIndexValid(arrIndex)) THEN

	moveLength := LastIndex - arrIndex;
	indexAdr := arr + arrIndex * _datatype.size;
	IF (moveLength = 0) THEN
		MEMSET(destAddr := indexAdr, fillByte := 16#00, n := _datatype.size);
	ELSE
		MEMMOVE(destAddr := indexAdr, srcAddr := indexAdr + _datatype.size, n := moveLength * _datatype.size);
		MEMSET(destAddr := indexAdr + moveLength * _datatype.size, fillByte := 16#00, n := _datatype.size);
	END_IF

	_length := _length - 1;
	
	IF (_length > 1 AND_THEN _length <= capacity / (GROWTH_FACTOR * 2)) THEN
		Shrink();
	END_IF
END_IF
END_METHOD


METHOD RemoveAll : List
VAR_INPUT
END_VAR

RemoveAll := THIS^;

__DELETE(arr);
_length := 0;

Alloc();
END_METHOD


METHOD Set : List
VAR_INPUT
	index	: INT; // Allow for indexing from end
	data	: ANY;
END_VAR
END_METHOD


METHOD PRIVATE Shrink : BOOL
VAR_INPUT
END_VAR
VAR
	sizeToCopy		: UDINT;
	allocSize		: UDINT;
	newArr			: PVOID;
END_VAR

capacity := capacity / GROWTH_FACTOR;
allocSize := _datatype.size * capacity;
newArr := __NEW(BYTE, allocSize);

sizeToCopy := _datatype.size * _length; 
MEMCPY(destAddr := newArr, srcAddr := arr, n := sizeToCopy);

__DELETE(arr);
arr := newArr;
END_METHOD

END_FUNCTION_BLOCK

// ---- Misc/P2WCHAR.TcPOU
FUNCTION P2WCHAR : WCHAR
VAR_INPUT
	p : POINTER TO WSTRING;
END_VAR
VAR
END_VAR

P2WCHAR := p^;

END_FUNCTION

// ---- Signal/Signal.TcPOU

FUNCTION Signal : REFERENCE TO SignalBundle
VAR_INPUT
	symbol			: REFERENCE TO BOOL;
END_VAR
VAR
END_VAR
VAR_STAT
	provider		: SignalProvider;
END_VAR


IF (__ISVALIDREF(symbol)) THEN
	Signal REF= provider.Get(symbol);
ELSE
	provider.Call();
END_IF

END_FUNCTION

// ---- Signal/SignalBundle.TcPOU

{attribute 'enable_dynamic_creation'}
FUNCTION_BLOCK SignalBundle
VAR_INPUT
END_VAR
VAR_OUTPUT
END_VAR
VAR		
	symbol				: REFERENCE TO BOOL;
	invertedLogic		: BOOL;
	
	_risingTrigger		: POINTER TO R_TRIG;
	_fallingTrigger		: POINTER TO F_TRIG;
	_timerOn			: POINTER TO TON;
	_timerOff			: POINTER TO TOF;
	_timerPulse			: POINTER TO TP;
	
	timerOnIO			: SignalTimer;
	timerOffIO			: SignalTimer;
	timerPulseIO		: SignalTimer;
	
	symbolVal			: BOOL;
END_VAR

METHOD Call : BOOL
VAR_INPUT
END_VAR
symbolVal := symbol XOR invertedLogic;

IF (_risingTrigger <> 0) THEN
	
	_risingTrigger^(CLK := symbolVal);
END_IF
IF (_fallingTrigger <> 0) THEN
	
	_fallingTrigger^(CLK := symbolVal);
END_IF
IF (_timerOn <> 0) THEN
	
	_timerOn^(IN := symbolVal);
END_IF
IF (_timerOff <> 0) THEN
	
	_timerOff^(IN := symbolVal);
END_IF
IF (_timerPulse <> 0) THEN
	
	_timerPulse^(IN := symbolVal);
END_IF
END_METHOD


PROPERTY fallingTrigger : REFERENCE TO BOOL
GET

IF (_fallingTrigger = 0) THEN
	
	_fallingTrigger := __NEW(F_TRIG);
END_IF

fallingTrigger REF= _fallingTrigger^.Q;
END_GET
END_PROPERTY


METHOD FB_exit : BOOL
VAR_INPUT
	bInCopyCode : BOOL; // if TRUE, the exit method is called for exiting an instance that is copied afterwards (online change).
END_VAR

IF (_risingTrigger <> 0) THEN
	
	__DELETE(_risingTrigger);
END_IF
IF (_fallingTrigger <> 0) THEN
	
	__DELETE(_fallingTrigger);
END_IF
IF (_timerOn <> 0) THEN
	
	__DELETE(_timerOn);
END_IF
IF (_timerOff <> 0) THEN
	
	__DELETE(_timerOff);
END_IF
IF (_timerPulse <> 0) THEN
	
	__DELETE(_timerPulse);
END_IF
END_METHOD


METHOD FB_init : BOOL
VAR_INPUT
	bInitRetains : BOOL; // if TRUE, the retain variables are initialized (warm start / cold start)
	bInCopyCode : BOOL;  // if TRUE, the instance afterwards gets moved into the copy code (online change)
	
	symbol			: REFERENCE TO BOOL; // Binded variable
	createAtStart	: STRING; // If strings RT, FT, TON, TOF, PT are found, then corresponding triggers or timers are created during init.
	invertedLogic	: BOOL; // Some variables (e.g. optical gates) may have inverted logic
END_VAR

THIS^.symbol REF= symbol;
THIS^.invertedLogic := invertedLogic;

IF (FIND(createAtStart, 'RT') > 0) THEN

	risingTrigger;
END_IF
IF (FIND(createAtStart, 'FT') > 0) THEN

	fallingTrigger;
END_IF
IF (FIND(createAtStart, 'TON') > 0) THEN

	timerOn;
END_IF
IF (FIND(createAtStart, 'TOF') > 0) THEN

	timerOff;
END_IF
IF (FIND(createAtStart, 'PT') > 0) THEN

	timerPulse;
END_IF
END_METHOD


PROPERTY risingTrigger : REFERENCE TO BOOL
GET

IF (_risingTrigger = 0) THEN
	
	_risingTrigger := __NEW(R_TRIG);
END_IF

risingTrigger REF= _risingTrigger^.Q;
END_GET
END_PROPERTY


PROPERTY timerOff : REFERENCE TO SignalTimer
GET

IF (_timerOff = 0) THEN
	
	_timerOff := __NEW(TOF);
	timerOffIO.PT REF= _timerOff^.PT;
	timerOffIO.ET REF= _timerOff^.ET;
	timerOffIO.Q REF= _timerOff^.Q;
END_IF

timerOff REF= timerOffIO;
END_GET
END_PROPERTY


PROPERTY timerOn : REFERENCE TO SignalTimer
GET

IF (_timerOn = 0) THEN
	
	_timerOn := __NEW(TON);
	timerOnIO.PT REF= _timerOn^.PT;
	timerOnIO.ET REF= _timerOn^.ET;
	timerOnIO.Q REF= _timerOn^.Q;
END_IF

timerOn REF= timerOnIO;
END_GET
END_PROPERTY


PROPERTY timerPulse : REFERENCE TO SignalTimer
GET

IF (_timerPulse = 0) THEN
	
	_timerPulse := __NEW(TP);
	timerPulseIO.PT REF= _timerPulse^.PT;
	timerPulseIO.ET REF= _timerPulse^.ET;
	timerPulseIO.Q REF= _timerPulse^.Q;
END_IF

timerPulse REF= timerPulseIO;
END_GET
END_PROPERTY

END_FUNCTION_BLOCK

// ---- Signal/SignalProvider.TcPOU

FUNCTION_BLOCK SignalProvider
VAR_INPUT
END_VAR
VAR_OUTPUT
END_VAR
VAR
	// hashtable of signals
	// register method creates new signal and saves pointer to hashtable
	// register and retrieve signal by its pointer
	
	mappings		: ARRAY[0..10] OF SignalMapping;
	count			: INT;
	lastMapping		: REFERENCE TO SignalMapping;
END_VAR


METHOD Call : BOOL
VAR_INPUT
END_VAR
VAR
	i		: INT;
END_VAR

FOR i := 0 TO count - 1 DO
	
	mappings[i].signal^.Call();
END_FOR
END_METHOD


METHOD FB_exit : BOOL
VAR_INPUT
	bInCopyCode : BOOL; // if TRUE, the exit method is called for exiting an instance that is copied afterwards (online change).
END_VAR
VAR
	i	: INT;
END_VAR

FOR i := 0 TO count DO
	
	__DELETE(mappings[i].signal);
END_FOR
END_METHOD


METHOD Find : INT
VAR_INPUT
	symbol	: REFERENCE TO BOOL;
END_VAR
VAR
	address	: POINTER TO SignalBundle;
	i		: INT;
END_VAR

Find := -1;

address := ADR(symbol);

FOR i := 0 TO count - 1 DO
	IF mappings[i].symbol = address THEN
		
		Find := i;

		RETURN;
	END_IF
END_FOR
END_METHOD


METHOD Get : REFERENCE TO SignalBundle
VAR_INPUT
	symbol	: REFERENCE TO BOOL;
END_VAR
VAR
	found	: INT;
END_VAR

found := Find(symbol);

IF (__ISVALIDREF(lastMapping) AND_THEN ADR(symbol) = lastMapping.symbol) THEN
	
	Get REF= lastMapping.signal^;
ELSIF (found = -1) THEN
	
	Get REF= Register(symbol, '', FALSE);
ELSE
	
	Get REF= mappings[found].signal^;
	lastMapping REF= mappings[found];
END_IF
END_METHOD


METHOD Register : REFERENCE TO SignalBundle
VAR_INPUT
	symbol	 		: REFERENCE TO BOOL;
	create			: STRING;
	inverted		: BOOL;
END_VAR

mappings[count].symbol := ADR(symbol); // Use the fact, that address of reference is address of the referenced variable
mappings[count].signal := __NEW(SignalBundle(symbol := symbol, createAtStart := create, invertedLogic := inverted));

Register REF= mappings[count].signal^;

lastMapping REF= mappings[count];

count := count + 1;
END_METHOD

END_FUNCTION_BLOCK

// ---- SimpleStepLogger/SimpleStepLogger.TcPOU
FUNCTION_BLOCK SimpleStepLogger
VAR_INPUT
END_VAR
VAR_OUTPUT
	logArray		: 	ARRAY[0..99] OF SimpleStepLog;
END_VAR
VAR
	count				: UINT;
	lastStepNumber		: LINT;
	stepWatch			: TON;
END_VAR

METHOD AutoLog : BOOL
VAR_INPUT
	step	: SimpleStepLog;
END_VAR
IF step.number <> lastStepNumber THEN
	LogStep(step);
	lastStepNumber := step.number;
END_IF
END_METHOD

METHOD FB_init : BOOL
VAR_INPUT
	bInitRetains : BOOL; // if TRUE, the retain variables are initialized (warm start / cold start)
	bInCopyCode : BOOL;  // if TRUE, the instance afterwards gets moved into the copy code (online change)
END_VAR
stepWatch(IN := TRUE, PT := DWORD_TO_TIME(16#FFFF_FFFF));
END_METHOD

METHOD LogStep : BOOL
VAR_INPUT
	step	: SimpleStepLog;
END_VAR
MEMMOVE(
	destAddr := ADR(logArray[1]),
	srcAddr := ADR(logArray[0]),
	n := SIZEOF(logArray[0]) * 99
);

logArray[0] := step;

IF count < 100 THEN
	
	count := count + 1;
END_IF
END_METHOD

END_FUNCTION_BLOCK

// ---- SymbolProvider/SymbolProvider_1.TcPOU

FUNCTION_BLOCK SymbolProvider_1
VAR_INPUT
END_VAR
VAR_OUTPUT
END_VAR
VAR
	symbolReader		: FB_JsonReadWriteDatatype;
END_VAR


METHOD GetDatatype : T_MaxString
VAR_INPUT
	symbol			: ANY;
END_VAR

GetDatatype := symbolReader.GetDatatypeNameByAddress(pData := symbol.pValue, nData := TO_UDINT(symbol.diSize));
END_METHOD


METHOD GetFullName : T_MaxString
VAR_INPUT
	symbol			: ANY;
END_VAR

GetFullName := symbolReader.GetSymbolNameByAddress(pData := symbol.pValue, nData := TO_UDINT(symbol.diSize));
END_METHOD


(* Returns full symbol name without its GVL or PRG name at the beginning
	example: for symbol 'MAIN.bStart' returns 'bStart'
*)
METHOD GetNameWithoutGlobalNameSpace : T_MaxString
VAR_INPUT
	symbol			: ANY;
END_VAR

GetNameWithoutGlobalNameSpace := symbolReader.GetSymbolNameByAddress(pData := symbol.pValue, nData := TO_UDINT(symbol.diSize));
GetNameWithoutGlobalNameSpace := RIGHT(STR := GetNameWithoutGlobalNameSpace, SIZE := LEN(GetNameWithoutGlobalNameSpace) - FIND(STR1 := GetNameWithoutGlobalNameSpace, STR2 := '.'));
END_METHOD

END_FUNCTION_BLOCK

// ---- Tools/WRegex.TcPOU
FUNCTION_BLOCK WRegex
VAR_INPUT
END_VAR
VAR_OUTPUT
END_VAR
VAR
END_VAR

//https://stackoverflow.com/questions/4040835/how-do-i-write-a-simple-regular-expression-pattern-matching-function-in-c-or-c

METHOD match : BOOL
VAR_INPUT
	pattern : WSTRING;
	text	: WSTRING;
END_VAR
match := wmatchP(ADR(pattern), ADR(text));
END_METHOD

METHOD PRIVATE wmatchHere : BOOL
VAR_INPUT
	pattern : POINTER TO WSTRING;
	text	: POINTER TO WSTRING;
END_VAR
IF P2WCHAR(pattern) = "$0000" THEN
	wmatchHere := TRUE;
	RETURN;
ELSIF P2WCHAR(pattern + 2) = "*" THEN
	wmatchHere := wmatchStar(P2WCHAR(pattern), pattern + 4, text);
	RETURN;
ELSIF P2WCHAR(pattern) = "$$" AND P2WCHAR(pattern + 2) = "$0000" THEN
	wmatchHere := P2WCHAR(text) = "$0000";
	RETURN;
ELSIF text^ <> "$0000" AND (P2WCHAR(pattern) = "." OR P2WCHAR(pattern) = P2WCHAR(text)) THEN
	wmatchHere := THIS^.wmatchHere(pattern + 2, text + 2);
	RETURN;
END_IF



///* matchhere: search FOR regexp AT beginning OF text */
//int matchhere(char *regexp, char *text)
//{
//    if (regexp[0] == '\0')
//        return 1;
//    if (regexp[1] == '*')
//        return matchstar(regexp[0], regexp+2, text);
//    if (regexp[0] == '$' && regexp[1] == '\0')
//        return *text == '\0';
//    if (*text!='\0' && (regexp[0]=='.' || regexp[0]==*text))
//        return matchhere(regexp+1, text+1);
//    return 0;
//}
END_METHOD

METHOD wmatchP : BOOL
VAR_INPUT
	pattern : POINTER TO WSTRING;
	text	: POINTER TO WSTRING;
END_VAR
IF P2WCHAR(pattern) = "^" THEN
	wmatchP := wmatchHere(pattern + 2, text);
END_IF
REPEAT
	IF wmatchHere(pattern, text) THEN
		wmatchP := TRUE;
		RETURN;
	END_IF
UNTIL
	NOT(P2WCHAR(text) <> "$0000") AND (text := text + 2) <> NULL //pointer dereference and increment oneliner
END_REPEAT


///* match: search FOR regexp anywhere in text */
//int match(char *regexp, char *text)
//{
//    if (regexp[0] == '^')
//        return matchhere(regexp+1, text);
//    do {    /* must look even if string is empty */
//        if (matchhere(regexp, text))
//            return 1;
//    } while (*text++ != '\0');
//    return 0;
//}
END_METHOD

METHOD PRIVATE wmatchStar : BOOL
VAR_INPUT
	c		: WCHAR;
	pattern : POINTER TO WSTRING;
	text	: POINTER TO WSTRING;
END_VAR
REPEAT
	IF wmatchHere(pattern, text) THEN
		wmatchStar := TRUE;
		RETURN;
	END_IF
UNTIL
	NOT(P2WCHAR(text) <> "$0000" AND (P2WCHAR(text) = c OR c = ".")) AND (text := text + 2) > null
END_REPEAT
wmatchStar := FALSE;


///* matchstar: search FOR c*regexp AT beginning OF text */
//int matchstar(int c, char *regexp, char *text)
//{
//    do {    /* a * matches zero or more instances */
//        if (matchhere(regexp, text))
//            return 1;
//    } while (*text != '\0' && (*text++ == c || c == '.'));
//    return 0;
//}
END_METHOD

END_FUNCTION_BLOCK
